INTERFACE I_OnCommand

PROPERTY IsOn : Bool
GET
END_GET
END_PROPERTY

METHOD On
END_METHOD

END_INTERFACE

(* stored: Version 1.1.0.1, ProductVersion 3.1.4024.12
   Itf I_OnCommand: Id {27cd863a-1f4c-4950-b003-e7bdb5d94782}
   Property IsOn: Id {5c96e1e8-b25a-4553-bca5-7b707f5765b7}
   Get Get: Id {f864fd32-8ac4-4544-976a-58440b1a7e94}
   Method On: Id {b8c07f9c-924a-422c-8bb6-74992f051256} *)
